(* Logix 5000 project; controller Test Emulate 5570 rev 30.12; software revision 30.00 *)

TASK MainTask (continuous, watchdog 500 ms) : MainProgram

MODULES
   Local : Emulate 5570 (ICP 2, rev 30.12)
END_MODULES

PROGRAM MainProgram   (* main routine MainRoutine *)
VAR
   Button : BOOL;
   FakeOutput : BOOL;
   Light : BOOL;
   OneShot : BOOL;
END_VAR

ROUTINE MainRoutine   (* ladder *)
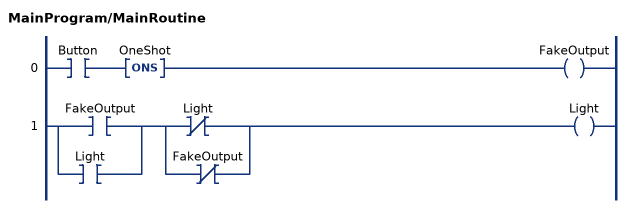
   0: XIC(Button)ONS(OneShot)OTE(FakeOutput);
   1: [XIC(FakeOutput) ,XIC(Light) ][XIO(Light) ,XIO(FakeOutput) ]OTE(Light);
END_ROUTINE
END_PROGRAM
